       #MyWord := W#0;
       #MyBoolsinWord[8] := #"OpMode_Auto";    //EPICSName: OpMode_Auto
       #MyBoolsinWord[9] := #"OpMode_Manual";    //EPICSName: OpMode_Manual
       #MyBoolsinWord[10] := #"OpMode_Forced";    //EPICSName: OpMode_Forced
       #MyBoolsinWord[11] := #"Opened";    //EPICSName: Opened
       #MyBoolsinWord[12] := #"Closed";    //EPICSName: Closed
       #MyBoolsinWord[13] := #"Solenoid";    //EPICSName: Solenoid
       #MyBoolsinWord[14] := #"Inhibit_Manual";    //EPICSName: Inhibit_Manual
       #MyBoolsinWord[15] := #"Inhibit_Force";    //EPICSName: Inhibit_Force
       #MyBoolsinWord[0] := #"Inhibit_Lock";    //EPICSName: Inhibit_Lock
       #MyBoolsinWord[1] := #"GroupInterlock";    //EPICSName: GroupInterlock
       #MyBoolsinWord[2] := #"StartInterlock";    //EPICSName: StartInterlock
       #MyBoolsinWord[3] := #"StopInterlock";    //EPICSName: StopInterlock
       #MyBoolsinWord[4] := #"EnableBlkOpen";    //EPICSName: EnableBlkOpen
       #MyBoolsinWord[5] := #"EnableBlkClose";    //EPICSName: EnableBlkClose
       #MyBoolsinWord[6] := #"EnableAutoBtn";    //EPICSName: EnableAutoBtn
       #MyBoolsinWord[7] := #"EnableManualBtn";    //EPICSName: EnableManualBtn
       "PLCToEPICS"."Word"[#PLCToEPICSDataBlockOffset + 14] := #MyWord;

       #MyWord := W#0;
       #MyBoolsinWord[8] := #"EnableForcedBtn";    //EPICSName: EnableForcedBtn
       #MyBoolsinWord[9] := #"NormallyOpen";    //EPICSName: NormallyOpen
       #MyBoolsinWord[10] := #"DevLocked";    //EPICSName: DevLocked
       #MyBoolsinWord[11] := #"LatchAlarm";    //EPICSName: LatchAlarm
       #MyBoolsinWord[12] := #"GroupAlarm";    //EPICSName: GroupAlarm
       "PLCToEPICS"."Word"[#PLCToEPICSDataBlockOffset + 15] := #MyWord;

    //********************************************
    //*************COMMAND VARIABLES**************
    //********************************************


       #MyWord := "EPICSToPLC"."Word"[#EPICSToPLCDataBlockOffset + 0];
       "EPICSToPLC"."Word"[#EPICSToPLCDataBlockOffset + 0] := 0;
       #"Cmd_Auto" := #MyBoolsinWord[8];    //EPICSName: Cmd_Auto
       #"Cmd_Manual" := #MyBoolsinWord[9];    //EPICSName: Cmd_Manual
       #"Cmd_Force" := #MyBoolsinWord[10];    //EPICSName: Cmd_Force
       #"Cmd_ManuOpen" := #MyBoolsinWord[11];    //EPICSName: Cmd_ManuOpen
       #"Cmd_ManuClose" := #MyBoolsinWord[12];    //EPICSName: Cmd_ManuClose
       #"Cmd_ForceOpen" := #MyBoolsinWord[13];    //EPICSName: Cmd_ForceOpen
       #"Cmd_ForceClose" := #MyBoolsinWord[14];    //EPICSName: Cmd_ForceClose
       #"Cmd_AckAlarm" := #MyBoolsinWord[15];    //EPICSName: Cmd_AckAlarm
       #"Cmd_ForceUnlock" := #MyBoolsinWord[0];    //EPICSName: Cmd_ForceUnlock
       #"Cmd_DevLock" := #MyBoolsinWord[1];    //EPICSName: Cmd_DevLock
       #"Cmd_DevUnlock" := #MyBoolsinWord[2];    //EPICSName: Cmd_DevUnlock

    //********************************************
    //************PARAMETER VARIABLES*************
    //********************************************


       #MyDInt	:= 0;
       #MyWordsinDint[0]	:= "EPICSToPLC"."Word"[#EPICSToPLCDataBlockOffset + 1];
       #MyWordsinDint[1]	:= "EPICSToPLC"."Word"[#EPICSToPLCDataBlockOffset + 2];
       #"P_Faceplate_LockID" := #MyDInt;    //EPICSName: P_Faceplate_LockID

       #MyDInt	:= 0;
       #MyWordsinDint[0]	:= "EPICSToPLC"."Word"[#EPICSToPLCDataBlockOffset + 3];
       #MyWordsinDint[1]	:= "EPICSToPLC"."Word"[#EPICSToPLCDataBlockOffset + 4];
       #"P_BlockIcon_LockID" := #MyDInt;    //EPICSName: P_BlockIcon_LockID

       #MyReal	:= 0.0;
       #MyWordsinReal[0]	:= "EPICSToPLC"."Word"[#EPICSToPLCDataBlockOffset + 5];
       #MyWordsinReal[1]	:= "EPICSToPLC"."Word"[#EPICSToPLCDataBlockOffset + 6];
       #"P_OpenSP" := #MyReal;    //EPICSName: P_OpenSP

       #MyReal	:= 0.0;
       #MyWordsinReal[0]	:= "EPICSToPLC"."Word"[#EPICSToPLCDataBlockOffset + 7];
       #MyWordsinReal[1]	:= "EPICSToPLC"."Word"[#EPICSToPLCDataBlockOffset + 8];
       #"P_CloseSP" := #MyReal;    //EPICSName: P_CloseSP
    Else
       #DEVICE_PARAM_OK := FALSE; //Invalid Hash
    END_IF;
END_FUNCTION_BLOCK

DATA_BLOCK "DEV_LabS-ICS:Cryo-PLC-163_iDB"
{ S7_Optimized_Access := 'TRUE' }
VERSION : 1.0
NON_RETAIN
"DEVTYPE_CMS_GLOBAL"
BEGIN
END_DATA_BLOCK


DATA_BLOCK "DEV_LabS-ICS:Cryo-LT-163_iDB"
{ S7_Optimized_Access := 'TRUE' }
VERSION : 1.0
NON_RETAIN
"DEVTYPE_ICS_PT"
BEGIN
END_DATA_BLOCK


DATA_BLOCK "DEV_LabS-ICS:Cryo-PT-163_iDB"
{ S7_Optimized_Access := 'TRUE' }
VERSION : 1.0
NON_RETAIN
"DEVTYPE_ICS_PT_MBAR"
BEGIN
END_DATA_BLOCK


DATA_BLOCK "DEV_LabS-ICS:Cryo-CV-090_iDB"
{ S7_Optimized_Access := 'TRUE' }
VERSION : 1.0
NON_RETAIN
"DEVTYPE_ICS_SCV"
BEGIN
END_DATA_BLOCK

FUNCTION "EPICS_device_calls" : Void
{ S7_Optimized_Access := 'TRUE' }
VERSION : 1.0

   VAR_TEMP
      "LabS-ICS:Cryo-PLC-163" : Bool;   // HASH codes are OK
      "LabS-ICS:Cryo-LT-163" : Bool;   // HASH codes are OK
      "LabS-ICS:Cryo-PT-163" : Bool;   // HASH codes are OK
      "LabS-ICS:Cryo-CV-090" : Bool;   // HASH codes are OK
   END_VAR

BEGIN
      //Author: Miklos Boros (miklos.boros@esss.se), Copyrigth 2017-2020 by European Spallation Source, Lund
      //This block was generated by PLCFactory
      //According to HASH:-819074987
      //Description: Description: This function calls the devices according to the corresponding device type

        //DO NOT Modify the following line!!!
        "Utilities".TestInProgress := FALSE;
        "Utilities".EPICS_Device_calls_precessed := TRUE;


        //********************************************
        // Device name: LabS-ICS:Cryo-PLC-163
        // Device type: CMS_GLOBAL
        //********************************************

      "DEV_LabS-ICS:Cryo-PLC-163_iDB" (EPICSToPLCLength:=17,
      EPICSToPLCDataBlockOffset:=10,
      PLCToEPICSLength:=53,
      PLCToEPICSDataBlockOffset:=10);

        //********************************************
        // Device name: LabS-ICS:Cryo-LT-163
        // Device type: ICS_PT
        //********************************************

      "DEV_LabS-ICS:Cryo-LT-163_iDB" (EPICSToPLCLength:=15,
      EPICSToPLCDataBlockOffset:=27,
      PLCToEPICSLength:=24,
      PLCToEPICSDataBlockOffset:=63);

        //********************************************
        // Device name: LabS-ICS:Cryo-PT-163
        // Device type: ICS_PT_MBAR
        //********************************************

      "DEV_LabS-ICS:Cryo-PT-163_iDB" (EPICSToPLCLength:=15,
      EPICSToPLCDataBlockOffset:=42,
      PLCToEPICSLength:=22,
      PLCToEPICSDataBlockOffset:=87);

        //********************************************
        // Device name: LabS-ICS:Cryo-CV-090
        // Device type: ICS_SCV
        //********************************************

      "DEV_LabS-ICS:Cryo-CV-090_iDB" (EPICSToPLCLength:=9,
      EPICSToPLCDataBlockOffset:=57,
      PLCToEPICSLength:=16,
      PLCToEPICSDataBlockOffset:=109);
END_FUNCTION
DATA_BLOCK "EPICS_DebuggerResult"
{ S7_Optimized_Access := 'TRUE' }
VERSION : 0.1
NON_RETAIN
   VAR
      EPICS_Debugger_UtilitiesCall : String;   // PLCFactory Utilities call status
      EPICS_Debugger_DeviceCalls : String;   // PLCFactory DeviceCalls status
      EPICS_Debugger_IOCHash : String;   // EPICS IOC Hash vs. PLCFactory Hash
      EPICS_Debugger_ModBusHeartBeat : String;   // EPICS IOC Modbus (IOC->PLC) communication status
      EPICS_Debugger_S7Connection : String;   // EPICS IOC S7 TCP (PLC->IOC) communication status
      EPICS_Debugger_EPICS_GeneralState : String;   // Main status of the EPICS IOC communication
      EPICS_S7Port : Int;   // Actual TCP port that has been opened by the PLC
      EPICS_ModbusPort : Int;   // Actual ModBusTCP port that has been opened by the PLC
      EPICS_PLC_EthernetInterface : UInt;   // The currently used HW Identifer of the Ethernet Port on the PLC dedicated to EPICS
      EPICS_PayloadSize_InBytes : UInt;   // The currently configured payload size in bytes
      EPICS_PLC_Hash : DInt;   // The PLC Hash
      EPICS_PLCFactory_Version : String;   // The PLCFactory version that was used to generate the PLC code
      EPICS_CommunicationOK : Bool;   // Overall EPICS communication is OK
   END_VAR

BEGIN

END_DATA_BLOCK
FUNCTION_BLOCK "EPICS_DebuggerFB"
{ S7_Optimized_Access := 'TRUE' }
VERSION : 0.1
   VAR
      CheckUtilitiesTON {OriginalPartName := 'IEC_TIMER'; LibVersion := '1.0'; ExternalAccessible := 'False'; ExternalVisible := 'False'; ExternalWritable := 'False'} : TON_TIME;
      UtilSquareErrorTON { ExternalAccessible := 'False'; ExternalVisible := 'False'; ExternalWritable := 'False'} : Bool;
      CheckUtilitiesTON2 {OriginalPartName := 'IEC_TIMER'; LibVersion := '1.0'; ExternalAccessible := 'False'; ExternalVisible := 'False'; ExternalWritable := 'False'} : TON_TIME;
      UtilSquareErrorTON2 { ExternalAccessible := 'False'; ExternalVisible := 'False'; ExternalWritable := 'False'} : Bool;
      ModBus_TON {OriginalPartName := 'IEC_TIMER'; LibVersion := '1.0'; ExternalAccessible := 'False'; ExternalVisible := 'False'; ExternalWritable := 'False'} : TON_TIME;
      ModBus_wordsave { ExternalAccessible := 'False'; ExternalVisible := 'False'; ExternalWritable := 'False'} : Word;
   END_VAR
   VAR DB_SPECIFIC
      Helper_String { ExternalAccessible := 'False'; ExternalVisible := 'False'; ExternalWritable := 'False'} : String;
      Helper_String_Array { ExternalAccessible := 'False'; ExternalVisible := 'False'; ExternalWritable := 'False'} AT Helper_String : Struct
         String_Maximal { ExternalAccessible := 'False'; ExternalVisible := 'False'; ExternalWritable := 'False'} : Byte;
         String_Actual { ExternalAccessible := 'False'; ExternalVisible := 'False'; ExternalWritable := 'False'} : Byte;
         StringValueArray { ExternalAccessible := 'False'; ExternalVisible := 'False'; ExternalWritable := 'False'} : Array[0..15] of Byte;
      END_STRUCT;
   END_VAR
   VAR
      S7ConnTON {OriginalPartName := 'IEC_TIMER'; LibVersion := '1.0'; ExternalAccessible := 'False'; ExternalVisible := 'False'; ExternalWritable := 'False'} : TON_TIME;
   END_VAR

   VAR_TEMP
      AllOK { ExternalAccessible := 'False'; ExternalVisible := 'False'; ExternalWritable := 'False'} : Bool;
      i : Int;
      ModBusOK : Bool;
      S7OK : Bool;
   END_VAR


BEGIN
	//Author: Miklos Boros (miklos.boros@esss.se), Copyrigth 2017-2020 by European Spallation Source, Lund
	//This block was generated by PLCFactory
	//Description: This FB checks the EPICS configuration and outputs the result into EPICS_DebuggerResult.

	//DO NOT Modify this block!!!

	//AllOK will be evaluated in this code and passed to the EPICS_CommunicationOK signal that can be used by the PLC logic
	#AllOK := TRUE;

	#CheckUtilitiesTON(IN:="Utilities".Square_100ms,
	                   PT:=T#200ms,
	                   Q=>#UtilSquareErrorTON);

	#CheckUtilitiesTON2(IN := NOT "Utilities".Square_100ms,
	                   PT := T#200ms,
	                   Q => #UtilSquareErrorTON2);


	#ModBus_TON(IN := #ModBus_wordsave = "EPICSToPLC"."Word"[2],
	            PT := T#5s);


     "EPICS_DebuggerResult".#EPICS_PayloadSize_InBytes := 250;
     "EPICS_DebuggerResult".#EPICS_PLC_Hash := -819074987;
     "EPICS_DebuggerResult".#EPICS_PLCFactory_Version := 'commitID';

	IF ("Utilities".AlwaysOn = FALSE) THEN
	    "EPICS_DebuggerResult".#EPICS_Debugger_UtilitiesCall := 'ERROR: FunctionBlock: "_UilitiesFB" is called with a wrong InstanceDB. Call it with the existing iDB named: "Utilities" AND check if the System Memory bits and the System Clock byte is enabled!';
         #AllOK := FALSE;
	ELSE
	    IF (#UtilSquareErrorTON OR #UtilSquareErrorTON2) THEN
	        "EPICS_DebuggerResult".#EPICS_Debugger_UtilitiesCall := 'ERROR: FunctionBlock: "_UilitiesFB" is called with a wrong InstanceDB. Call it with the existing iDB named: "Utilities" AND check if the System Memory bits and the System Clock byte is enabled!';
             #AllOK := FALSE;
	    ELSE
	        "EPICS_DebuggerResult".#EPICS_Debugger_UtilitiesCall := 'OK: EPICS Utilities works as expected.';

	    END_IF;
	END_IF;

	IF ("Utilities".EPICS_Device_calls_precessed) THEN
	    "EPICS_DebuggerResult".#EPICS_Debugger_DeviceCalls := 'OK: "EPICS_device_calls" is called as expected.';
	ELSE
	    "EPICS_DebuggerResult".#EPICS_Debugger_DeviceCalls := 'ERROR: "EPICS_device_calls" is not called in OB1!';
         #AllOK := FALSE;
	END_IF;

	IF (("EPICSToPLC"."Word"[0] = "PLCToEPICS"."Word"[0]) AND ("EPICSToPLC"."Word"[1] = "PLCToEPICS"."Word"[1])) THEN
	    "EPICS_DebuggerResult".#EPICS_Debugger_IOCHash := 'OK: IOC and PLC hash are equal.';
	ELSE
	    "EPICS_DebuggerResult".#EPICS_Debugger_IOCHash := 'ERROR: IOC and PLC hash are NOT equal!';
         #AllOK := FALSE;
	END_IF;

	IF (#ModBus_TON.Q) THEN
	    "EPICS_DebuggerResult".#EPICS_Debugger_ModBusHeartBeat := 'ERROR: The IOC is not sending any HeartBeat via ModBus!';
         #AllOK := FALSE;
	    #ModBusOK := FALSE;
	ELSE
	    "EPICS_DebuggerResult".#EPICS_Debugger_ModBusHeartBeat := 'OK: ModBus HeartBeat is received as expected.';
	    #ModBusOK := TRUE;
	END_IF;

	#S7ConnTON(IN := NOT "_CommsPLC_EPICS_DB".SendDone, PT := T#3s);

	IF ("_CommsPLC_EPICS_DB".BytesToSend > 0) THEN

	    IF (#S7ConnTON.Q) THEN
	        "EPICS_DebuggerResult".EPICS_Debugger_S7Connection := 'ERROR: EPICS S7 connection can not send Status variables!';
	        #S7OK := FALSE;
             #AllOK := FALSE;
	    ELSE
	        "EPICS_DebuggerResult".EPICS_Debugger_S7Connection := 'OK: EPICS S7 works as expected.';
	        #S7OK := TRUE;

	    END_IF;
	ELSE
	    "EPICS_DebuggerResult".EPICS_Debugger_S7Connection := 'OK: EPICS S7 disabled, there is no Status variable to send.';
	    #S7OK := TRUE;
	END_IF;

	IF (#ModBusOK AND #S7OK) THEN
	    "EPICS_DebuggerResult".EPICS_Debugger_EPICS_GeneralState := 'OK. EPICS IOC communication is ONLINE.';
	END_IF;

	IF (#ModBusOK AND NOT #S7OK) THEN
	    "EPICS_DebuggerResult".EPICS_Debugger_EPICS_GeneralState := 'ERROR. ModBus seems to be working but S7 TCP is blocked. Try to check your PLC router IP.';
         #AllOK := FALSE;
	END_IF;

	IF (NOT #ModBusOK AND #S7OK) THEN
	    "EPICS_DebuggerResult".EPICS_Debugger_EPICS_GeneralState := 'ERROR. ModBus seems to be offline. Waiting for IOC to finish connecting to the PLC.';
         #AllOK := FALSE;
	END_IF;

	IF ( NOT #ModBusOK AND NOT #S7OK) THEN
	    "EPICS_DebuggerResult".EPICS_Debugger_EPICS_GeneralState := 'ERROR. Both ModBus and S7 TCP seems to be offline. Check if your IOC is running and if it is connected to the right PLC interface. Your HardwareID comes from CCDB!';
         #AllOK := FALSE;
	END_IF;

	"EPICS_DebuggerResult".EPICS_ModbusPort := "_CommsPLC_EPICS_DB".MBPort;
	"EPICS_DebuggerResult".EPICS_S7Port := "_CommsPLC_EPICS_DB".S7Port;
	"EPICS_DebuggerResult".EPICS_PLC_EthernetInterface :=  "_CommsPLC_EPICS_DB".InterfaceID;

	#ModBus_wordsave := "EPICSToPLC"."Word"[2];

	//Put the Overall result to the Globl DB
	"EPICS_DebuggerResult".EPICS_CommunicationOK := #AllOK;


END_FUNCTION_BLOCK
DATA_BLOCK "EPICS_DebuggerFB_iDB"
{ S7_Optimized_Access := 'TRUE' }
VERSION : 0.1
NON_RETAIN
"EPICS_DebuggerFB"

BEGIN

END_DATA_BLOCK
ORGANIZATION_BLOCK "EPICS_DebuggerOB"
TITLE = "Main Program Sweep (Cycle)"
{ S7_Optimized_Access := 'TRUE' }
VERSION : 0.1

BEGIN
	//Author: Miklos Boros (miklos.boros@esss.se), Copyrigth 2017-2020 by European Spallation Source, Lund
	//This block was generated by PLCFactory
	//Description: This OB is a cyclic OB called in every PLC cycle and EPICS_DebuggerFB checks the EPICS configuration.

	//DO NOT Modify this block!!!
	"EPICS_DebuggerFB_iDB"();


END_ORGANIZATION_BLOCK
DATA_BLOCK "EPICSToPLC"
{ S7_Optimized_Access := 'FALSE' }
VERSION : 0.1
//########## EPICS->PLC datablock ##########
   STRUCT
      "Word" { ExternalAccessible := 'False'; ExternalVisible := 'False'; ExternalWritable := 'False'; } : Array[0..65] of Word;
   END_STRUCT;

BEGIN

END_DATA_BLOCK

DATA_BLOCK "PLCToEPICS"
{ S7_Optimized_Access := 'FALSE' }
VERSION : 0.1
NON_RETAIN
//########## PLC->EPICS datablock ##########
   STRUCT
      "Word" { ExternalAccessible := 'False'; ExternalVisible := 'False'; ExternalWritable := 'False'; } : Array[0..124] of Word;
   END_STRUCT;

BEGIN

END_DATA_BLOCK

FUNCTION "_CommsEPICS" : Void
{ S7_Optimized_Access := 'TRUE' }
VERSION : 0.1
   VAR_TEMP
      PLC_Hash : DInt;
   END_VAR

BEGIN
	//Heartbeat PLC->EPICS
	IF "Utilities".Pulse_1s THEN
	    "PLCToEPICS"."Word"[2] := "PLCToEPICS"."Word"[2] + 1;
	    IF "PLCToEPICS"."Word"[2] >= 32000 THEN
	        "PLCToEPICS"."Word"[2] := 0;
	    END_IF;
	END_IF;

	// PLC Factory commit ID: commitID
	// PLC Hash (Generated by PLC Factory)
	#PLC_Hash := DINT#-819074987;

	// Send the PLC Hash to the EPICS IOC
	"PLCToEPICS"."Word"[1] := DINT_TO_WORD(#PLC_Hash);
	"PLCToEPICS"."Word"[0] := DINT_TO_WORD(SHR(IN := #PLC_Hash, N := 16));

	// Send the PLC parameter upload status to the EPICS IOC
	"PLCToEPICS"."Word"[3] := "EPICSToPLC"."Word"[5];
     "Utilities".EPICSParametersStatus := "EPICSToPLC"."Word"[5];

	// Put the PLC Hash into the Modbus map
	"EPICSToPLC"."Word"[4] := DINT_TO_WORD(#PLC_Hash);
	"EPICSToPLC"."Word"[3] := DINT_TO_WORD(SHR(IN := #PLC_Hash, N := 16));


	// Put the payload size (in bytes) into the Modbus map
	"EPICSToPLC"."Word"[6] := 250;

	// Call the comms block to provide PLC<->EPICS comms
	"_CommsPLC_EPICS_DB"(Enable         := "Utilities".AlwaysOn,
	                     SendTrigger    := "Utilities".Pulse_200ms,
	                     BytesToSend    := 250,
	                     InterfaceID    := 0,
	                     S7ConnectionID := 256,
	                     MBConnectionID := 255,
	                     S7Port         := 2000,
	                     MBPort         := 502,
	                     PLCToEPICSData := "PLCToEPICS"."Word",
	                     EPICSToPLCData := "EPICSToPLC"."Word");

END_FUNCTION
